// TIA Portal project "S7-1500 ile Trafik Lambası Uygulaması" (V18)

(* hardware
DEVICE "S7-1500/ET200MP station_1"  S7-1500 station
   slot 0: "Rail_0"  Rack  6ES7 590-1***0-0AA0
   slot 1: "PLC_1"  CPU 1512C-1 PN  6ES7 512-1CK01-0AB0  V2.8
      slot 3: "CPU display_1"  6ES7591-1AA00-0AA0
      slot 32768: "PROFINET interface_1"  X1
         slot 32769: "Port_1"  X1 P1
         slot 32770: "Port_2"  X1 P2
      slot 34817: "Virtual CP interface port_1"  Virtual CP interface port  Virtual CP interface port
DEVICE "HMI_1"  KTP700 Basic PN
   slot 0: "HMI_1"  KTP700 Basic PN  6AV2 123-2GB03-0AX0  14.0.1.0
   slot 1: "HMI_RT_1"  KTP700 Basic PN  6AV2 123-2GB03-0AX0  14.0.1.0
   slot 5: "HMI_1.IE_CP_1"  PROFINET Interface  14.0.1.0
      slot 1: "PROFINET Interface_1"  PROFINET Interface
         slot 1: "Port_1"  Port
*)

// ===== PLC "PLC_1"  CPU 1512C-1 PN =====

VAR_GLOBAL   // PLC tag table "Default tag table"
   "Stop" AT %M0.0 : Bool;
   "Start" AT %M0.1 : Bool;
   "Kırmızı" AT %Q0.0 : Bool;
   "Sarı" AT %Q0.1 : Bool;
   "Yeşil" AT %Q0.2 : Bool;
   "Döngü" AT %M0.5 : Bool;
   "Zaman Değeri" AT %MD100 : Time;
   "Zamanlayıcı Reset" AT %M0.7 : Bool;
   "Zamanlayıcı (Saniye)" AT %MD120 : DInt;
   "Tag_1" AT %M0.6 : Bool;
   "Zaman(Saniye)" AT %MD200 : DInt;
   "Tag_2" AT %M1.1 : Bool;
END_VAR

// folder: System blocks/Program resources

DATA_BLOCK "Zamanlayıcı"   // DB5
{ S7_Optimized_Access := 'TRUE' }
AUTHOR : Simatic
FAMILY : IEC
NAME : IEC_TMR
VERSION : 1.0
// stored: InstanceOfName IEC_TIMER
"IEC_TIMER"
BEGIN
END_DATA_BLOCK

// folder: (top level)

ORGANIZATION_BLOCK "Main"   // OB1, LAD, ProgramCycle
TITLE = "Main Program Sweep (Cycle)"
{ S7_Optimized_Access := 'TRUE' }
VERSION : 0.1
   VAR_INPUT
      Initial_Call : Bool;   // Initial call of this OB
      Remanence : Bool;   // =True, if remanent data are available
   END_VAR
   VAR_TEMP   // added for the SCL form of the ladder/FBD networks
      _w1 : Bool;
   END_VAR
BEGIN

REGION Network 1: Trafik Lambası
   // Starta basınca;
   // kırmızı 12s
   // Kırmızı+sarı 3s
   // Yeşil 10s
   // Sarı 3s
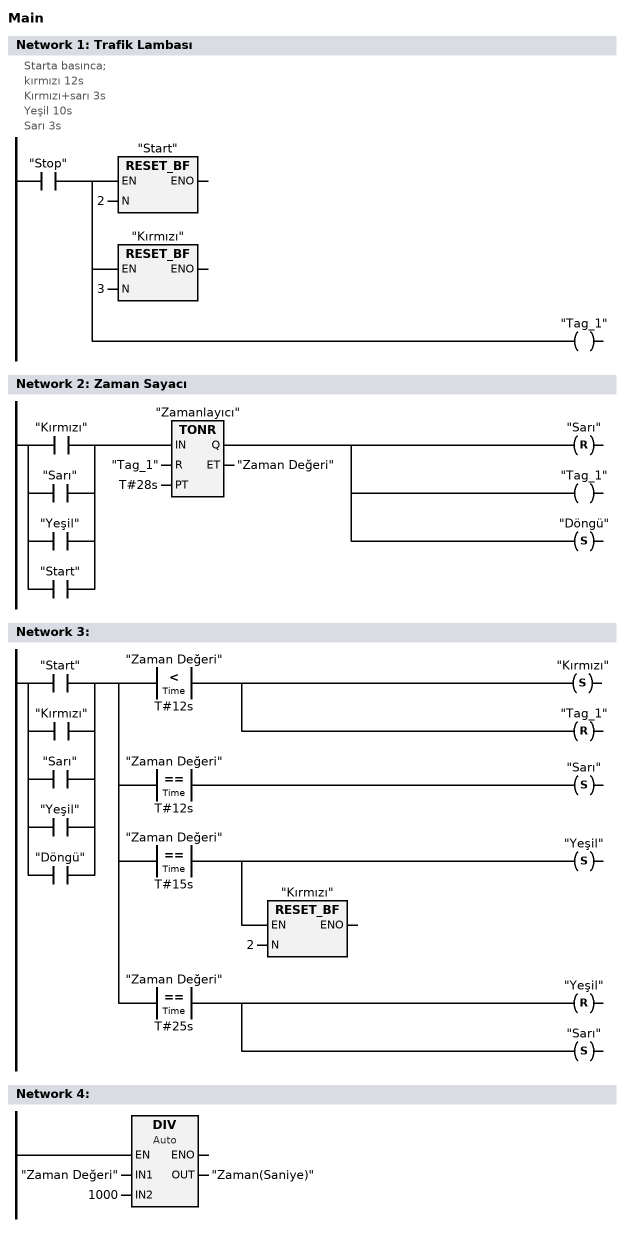
   // no SCL statement known for RBitfield: written as a call
   #_w1 := "Stop";
   IF #_w1 THEN
       RESET_BF(operand := "Start", n := 2);
       RESET_BF(operand := "Kırmızı", n := 3);
   END_IF;
   "Tag_1" := #_w1;
END_REGION

REGION Network 2: Zaman Sayacı
   "Zamanlayıcı".TONR(IN := "Kırmızı" OR "Sarı" OR "Yeşil" OR "Start",
                      R := "Tag_1",
                      PT := T#28s,
                      ET => "Zaman Değeri");
   IF "Zamanlayıcı".Q THEN "Sarı" := FALSE; END_IF;
   "Tag_1" := "Zamanlayıcı".Q;
   IF "Zamanlayıcı".Q THEN "Döngü" := TRUE; END_IF;
END_REGION

REGION Network 3
   // no SCL statement known for RBitfield: written as a call
   #_w1 := "Start" OR "Kırmızı" OR "Sarı" OR "Yeşil" OR "Döngü";
   IF #_w1 AND ("Zaman Değeri" < T#12s) THEN
       "Kırmızı" := TRUE;
       "Tag_1" := FALSE;
   END_IF;
   IF #_w1 AND ("Zaman Değeri" = T#12s) THEN "Sarı" := TRUE; END_IF;
   IF #_w1 AND ("Zaman Değeri" = T#15s) THEN
       "Yeşil" := TRUE;
       RESET_BF(operand := "Kırmızı", n := 2);
   END_IF;
   IF #_w1 AND ("Zaman Değeri" = T#25s) THEN
       "Yeşil" := FALSE;
       "Sarı" := TRUE;
   END_IF;
END_REGION

REGION Network 4
   RUNG wire#powerrail
      Div(in1 := "Zaman Değeri", in2 := 1000, out => "Zaman(Saniye)")
   END_RUNG
   // the same network as SCL:
   "Zaman(Saniye)" := "Zaman Değeri" / 1000;
END_REGION
END_ORGANIZATION_BLOCK

(* ===== HMI "HMI_RT_1" =====
system functions are stored by id; their names below are inferred from use
connection "Connection_1": ETHERNET, SMART_S7_1500_OMS
connection "HMI_Connection_1": ETHERNET, SMART_S7_1500_OMS

HMI tags "Default tag table"
   "Tag_ScreenNumber" : UInt, internal
   "Start_1" : Bool = PLC Start AT %M0.1, 100 ms
   "Kırmızı" : Bool = PLC Kırmızı AT %Q0.0, 100 ms
   "Sarı" : Bool = PLC Sarı AT %Q0.1, 100 ms
   "Yeşil" : Bool = PLC Yeşil AT %Q0.2, 100 ms
   "Stop" : Bool = PLC Stop AT %M0.0, 100 ms
   "Tag_4" : Time = PLC "Zaman Değeri" AT %MD100, 100 ms
   "Tag_2" : DInt = PLC "Zaman(Saniye)" AT %MD200, 100 ms

graphic list "Geri Hareket": 0 'Graphic_22'; 1 'Graphic_23'

graphic list "İleri Hareket": 0 'Graphic_21'; 1 'Graphic_20'

Template "Template_1" 800x480
   Button "Exit" at 714,429 size 71x50; TextOff 'Exit'; PictureOff "ExitRuntime_KTP700_Basic_PN_TR"; PictureOn "ExitRuntime_KTP700_Basic_PN_TR"
      on Release: StopRuntime(0)
   Button "Language" at 614,429 size 71x50; TextOff 'Language'; PictureOff "ToggleLanguage_KTP700_Basic_PN_TR"; PictureOn "ToggleLanguage_KTP700_Basic_PN_TR"
      on Release: function_fb9197e8(-1)
   Button "Log on" at 514,429 size 71x50; TextOff 'Log on'; PictureOff "Login_KTP700_Basic_PN_TR"; PictureOn "Login_KTP700_Basic_PN_TR"
      on Release: function_a2a04561()
   Button "Alarms" at 114,429 size 71x50; TextOff 'Alarms'; PictureOff "AlarmDisplay_KTP700_Basic_PN_TR"; PictureOn "AlarmDisplay_KTP700_Basic_PN_TR"
      on Release: function_ef3f5d25("Alarm window_Unacknowledged", -1)
   Button "Start screen" at 14,429 size 71x50; TextOff 'Start screen'; PictureOff "NavigateHome_KTP700_Basic_PN_TR"; PictureOn "NavigateHome_KTP700_Basic_PN_TR"
      on Release: ActivateScreen("Root screen", 0)
   SymbolicIOField "Symbolic_IO_Field_Screen" at 93,9 size 600x33; TextOff '0'; TextOn '1'; TextList "TextList_ScreenNames"
      ProcessValue <- "Tag_ScreenNumber"
      on Change: ActivateScreenByNumber("Tag_ScreenNumber", 0)
   DateTimeField "HmiScreenItemData" at 695,25 size 105x25
   DateTimeField "HmiScreenItemData_1" at 695,0 size 105x25
   GraphicView "Logo" at 0,0 size 91x51; Picture "Logo of HMI_1"

screen "Root screen" 800x480, template "Template_1"
   on GenerateScreen: SetTag("Tag_ScreenNumber", 1)
   Button "Button_4" at 432,80 size 129x50; TextOff 'Start'
      on Click: InvertBit("Start_1")
   Circle "Circle_1" at 316,93 size 52x52
      Appearance <- "Kırmızı"
   Circle "Circle_2" at 316,214 size 52x52
      Appearance <- "Yeşil"
   Circle "Circle_3" at 316,154 size 52x52
      Appearance <- "Sarı"
   Button "Button_1" at 432,136 size 129x50; TextOff 'Stop'
      on Press: SetBit("Stop")
      on Release: ResetBit("Stop")
   IOField "I/O field_1" at 432,195 size 129x54; FormatPattern s9999999999
      ProcessValue <- "Tag_2"
   TextField "Text field_1" at 129,113 size 146x23; Text '12 Saniye Kırmızı'
   TextField "Text field_2" at 164,172 size 111x23; Text '3 Saniye Sarı'
   TextField "Text field_3" at 147,226 size 128x23; Text '10 Saniye Yeşil'
*)